(* Logix 5000 project; controller EuniceF_ICA13 vendor 1 type 14 code 150 rev 37.11; software revision 37.00 *)

TASK MainTask (continuous, watchdog 500 ms) : MainProgram

MODULES
   Local : vendor 1 type 14 code 150 (Compact 0, rev 37.11)
      Discrete_IO : Embedded (Compact 1, rev 3.1, Output RPI 20 ms)
      Analog_IO : Embedded (Compact 2, rev 1.1, Output RPI 80 ms)
      Counters : Embedded (Compact 3, rev 1.1, Output RPI 20 ms)
END_MODULES

VAR_GLOBAL   (* controller tags *)
   Counter : COUNTER := (PRE := 20);
   Counter2 : COUNTER := (PRE := 20);
   Lot_Empty : BOOL;
   Lot_Full : BOOL;
   MyTotalCount : DINT;
   Toggle1 : BOOL;
   Toggle2 : BOOL;
END_VAR

PROGRAM MainProgram   (* main routine MainRoutine *)
VAR
   Counter1 : COUNTER;
   Toggle : BOOL;
END_VAR

ROUTINE MainRoutine   (* ladder *)
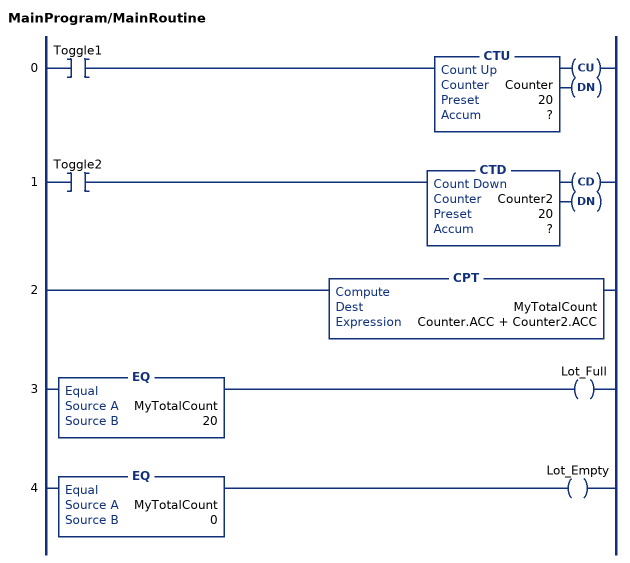
   0: XIC(Toggle1)CTU(Counter,?,?);
   1: XIC(Toggle2)CTD(Counter2,?,?);
   2: CPT(MyTotalCount,Counter.ACC + Counter2.ACC);
   3: EQ(MyTotalCount,20)OTE(Lot_Full);
   4: EQ(MyTotalCount,0)OTE(Lot_Empty);
END_ROUTINE
END_PROGRAM
